TYPE ST_Encoder :
STRUCT
	xENC_PWR_SW : BOOL;
	xENC_PWR : BOOL;
END_STRUCT
END_TYPE

(* stored: Version 1.1.0.1, ProductVersion 3.1.0.24
   DUT ST_Encoder: Id {bb2fe342-da49-4c90-9bde-8a4b26ef679c} *)
